// TIA Portal V21 export
DATA_BLOCK "DoManualModeDb"   // DB2
{ S7_Optimized_Access := 'FALSE' }
// stored: AutoNumber false
   VAR
      Mm01Cmd : Bool;
      Cp01Cmd : Bool;
      Htr : Bool;
      Lf01 : Bool;
      DoSpare1 : Bool;
      DoSpare2 : Bool;
      DoSpare3 : Bool;
      DoSpare4 : Bool;
      DoSpare5 : Bool;
      DoSpare6 : Bool;
   END_VAR
BEGIN
END_DATA_BLOCK
